TYPE T_ASTRO_COORDINATES :
STRUCT
	alpha: LREAL := 0;		// [hms]
	delta: LREAL := 0;		// [dms]
END_STRUCT
END_TYPE

(* stored: Version 1.1.0.1, ProductVersion 3.1.4024.10
   DUT T_ASTRO_COORDINATES: Id {db2983eb-a509-4f0b-b5de-2303464972df} *)
